// TIA Portal V17 export
// export: Created 2024-10-17T14:16:17.6196001Z, ExportSetting WithDefaults, DisplayName Totally Integrated Automation Portal, DisplayVersion V17 Update 4, DisplayName TIA Portal Openness, DisplayVersion V17 Update 4, DisplayName TIA Portal Version Control Interface, DisplayVersion V17, DisplayName SINAMICS Startdrive Advanced, DisplayVersion V17 Update2, DisplayName SINAMICS Startdrive G130, G150, S120, S150, SINAMICS MV, S210, DisplayVersion V17 Update2, DisplayName SINAMICS Startdrive G110M, G120, G120C, G120D, G120P, G115D, DisplayVersion V17 Update2, DisplayName STEP 7 Professional, DisplayVersion V17 Update 4, DisplayName STEP 7 Safety, DisplayVersion V17, DisplayName WinCC Advanced / Unified PC, DisplayVersion V17 Update 4
TYPE "LPMLV2022_typeEquipmentInterlock"
TITLE = LPMLV2022_typeEquipmentInterlock
// Support: tech.team.motioncontrol@siemens.com
// stored: IsFailsafeCompliant false
   STRUCT
      Blocked { ExternalWritable := 'False'} : Bool;   // Indicator for Unit/Machine Blocked. This bit, when set to 1, indicates that a downstream system is not able to accept product. In this condition, the equipment is capable of producing product but is in a suspended state due to a downstream system
      Starved { ExternalWritable := 'False'} : Bool;   // Indicator for Unit/Machine Starved. This bit, when set to 1, indicates that an upstream system is not able to supply product. In this condition, the equipment is capable of producing product but is in a suspended state due to an upstream system
   END_STRUCT;
END_TYPE
